//Calculate the number of Device
IF NOT bNumberIsCalculatet THEN
	IF diActualNumberOfDevices < diMaxNumberOfDevices THEN diNumberForThisDevice := diActualNumberOfDevices + 1; bNumberIsCalculatet := TRUE; END_IF 
		diNumberOfTotalDevices := diActualNumberOfDevices + 1;
			FPCalculatet.CLK := TRUE;
				diNumberForThisDevice := LIMIT(0,diNumberForThisDevice,diMaxNumberOfDevices);		
END_IF 
	//Reset when we have a online change
	IF bOnlineChange THEN bOnlineChange := FALSE; END_IF
		IF udiCounterOnlineChange <> udiCounterOnlineChange_CP THEN
			bNumberIsCalculatet := FALSE;
				diNumberForThisDevice := 0;
					diNumberOfTotalDevices := diNumberForThisDevice;
						udiCounterOnlineChange_CP := udiCounterOnlineChange;   
							bOnlineChange := TRUE;	
								FPCalculatet.CLK := FALSE;			
		END_IF  
		
FPCalculatet(CLK:= , Q=> bFPNumberIsCalculatet);

END_FUNCTION_BLOCK

// ---- Persistent Data/FBs Internal/PD Slave/FB_PersistentData_String.TcPOU
{attribute 'hide_all_locals'}
{attribute 'conditionalshow'}
FUNCTION_BLOCK FB_PersistentData_String
VAR_INPUT
	{attribute 'hide'}
	sText								: STRING(255);			//Actual Input Text						
END_VAR
VAR_OUTPUT
	{attribute 'hide'}
	bEventBasedActive					: BOOL;					//Event based saving is active
END_VAR
VAR
	sText_CP							: STRING(255);			//Text to compare the input Text
	fbTaskIndex							: GETCURTASKINDEX;		//Get the Task index
END_VAR

//Creator : Kai Ebensperger
//Company : Lynus AG
//Date : 15.02.2021
//Version : 1.0.0.0

//With this Function we can check if the Value on the Input of the Function ha changed an chan start to saving the persistent Data in Event Based Mode
//Work only with String Fromat
//Max 255 characters

//---------------------------------------------------------------Logic to start the save process---------------------------------------------------------------------------------------

bEventBasedActive := GVL_Persistent_Data.bEventBasedActive;

//After Restart the System set the Variables direct to actual value because they are loadet from the card
fbTaskIndex(index=> );
	IF TwinCAT_SystemInfoVarList._TaskInfo[fbTaskIndex.index].FirstCycle THEN sText_CP := sText; END_IF

IF NOT GVL_Persistent_Data.bBusy AND bEventBasedActive AND MEMCMP(ADR(sText),ADR(sText_CP),SIZEOF(sText_CP)) <> 0 THEN
	GVL_Persistent_Data.bSaveData := TRUE;
		sText_CP := sText;
END_IF

END_FUNCTION_BLOCK

// ---- Sensors/FBs Internal/Temperature/FB_Config_KL320x.TcPOU
{attribute 'conditionalshow'}
FUNCTION_BLOCK FB_Config_KL320x
VAR_INPUT
	{attribute 'hide'}
	eChooseSensorType		: E_ChooseSensortype_KL320x;			//Tel what sensor type is configred on the terminal
	{attribute 'hide'}
	iTimeout				: INT;									//Delay for timeout in seconds
	{attribute 'hide'}
	bWriteConfig			: BOOL;									//Positive edge start the sensor type configuration on the terminal
	{attribute 'hide'}
	bReadConfig				: BOOL;									//Posistive edge read out the actual configuration from the terminal
END_VAR
VAR_OUTPUT
	{attribute 'hide'}
	bConfigModeAktiv		: BOOL;									//True when the configuration mode is active
	{attribute 'hide'}
	bError					: BOOL;									//Error Bit
	{attribute 'hide'}
	b2Wire					: BOOL;									//Terminal is configured in the 2 wire mode
	{attribute 'hide'}
	iRawValueTerminal		: INT;									//Raw value from the terminal when the configuration mode is done
	{attribute 'hide'}
	usiState				: USINT;								//State from the KL320x terminal
	{attribute 'hide'}
	sSensorType				: STRING(50);							//Configured sensortype as string after read out the configuration
END_VAR
VAR
	{attribute 'hide'}
	FP0						: R_TRIG;								//Internal positive edge
	{attribute 'hide'}
	FP1						: R_TRIG;								//Internal positive edge
	{attribute 'hide'}
	timTimout				: TON;									//Timer for timeout
	{attribute 'hide'}
	eStep					: E_Step_Config_Terminal_KL320x;		//Step terminal configuration
	stDataIn		AT%I*	: ST_InputData_KL320x;					//Input Data from the KL320x
	stDataOut		AT%Q*	: ST_OutputData_KL320x;					//Output Data from the KL320x
	{attribute 'hide'}
	bCheck					: BOOL;									//True after the value is writen in the register
END_VAR

//Creator : Kai Ebensperger
//Company : Lynus AG
//Date : 02.06.2021
//Version : 1.0.0.0

//This function block is used to configure a KL3201, KL3202 and KL3204
//Communicate about the input and output Data from the terminal
//Attention : A KL3208 cannot be configured with this function block

(*---------------------------------------------------------------Check the limits of the inputs-------------------------------------------------------------------------------*)

iTimeout := LIMIT(1,iTimeout,10);

(*---------------------------------------------------------------Start the configuration or read out the actual configuration-------------------------------------------------------------------------------*)

FP0(CLK:= bWriteConfig, Q=> );
	FP1(CLK:= bReadConfig, Q=> );

	IF FP0.Q AND NOT bConfigModeAktiv THEN
		eStep := E_Step_Config_Terminal_KL320x.eRegister31DeactivateWriteProtection_KL320x;
	END_IF
		IF FP1.Q AND NOT bConfigModeAktiv THEN
			eStep := E_Step_Config_Terminal_KL320x.eReadConfiguration_KL320x;
		END_IF
	
CASE eStep OF
		
	E_Step_Config_Terminal_KL320x.eInit_KL320x: //Init Step						
										
		iRawValueTerminal := stDataIn.iDataIn;
			usiState := stDataIn.usiState;
				stDataOut.iDataOut := 0;
					stDataOut.usiControl := 0;
						bConfigModeAktiv := FALSE;
							timTimout.IN := FALSE;
								bCheck := FALSE;
			
	E_Step_Config_Terminal_KL320x.eRegister31DeactivateWriteProtection_KL320x: //Deactivate Write protecton on register 31 to write data on other registers			
													
		bConfigModeAktiv := TRUE;
			timTimout.IN := TRUE;
				bError := FALSE;
							
					IF NOT bCheck THEN	
						stDataOut.usiControl.0 := TRUE;
							stDataOut.usiControl.1 := TRUE;
								stDataOut.usiControl.2 := TRUE;
									stDataOut.usiControl.3 := TRUE;
										stDataOut.usiControl.4 := TRUE;
											stDataOut.usiControl.5 := FALSE;				
												stDataOut.usiControl.6 := TRUE;
													stDataOut.usiControl.7 := TRUE;
						END_IF
														
							//Activate the code in register 31
							stDataOut.iDataOut := 16#1235;
		
							//Feedback from the input data from the terminal
							IF stDataIn.iDataIn.0 = FALSE AND
								stDataIn.iDataIn.1 = FALSE AND
									stDataIn.iDataIn.2 = FALSE AND
										stDataIn.iDataIn.3 = FALSE AND
											stDataIn.iDataIn.4 = FALSE AND
												stDataIn.iDataIn.5 = FALSE AND
													stDataIn.iDataIn.6 = FALSE AND
														stDataIn.iDataIn.7 = FALSE AND
															stDataIn.iDataIn.8 = FALSE AND
																stDataIn.iDataIn.9 = FALSE AND
																	stDataIn.iDataIn.10 = FALSE AND
																		stDataIn.iDataIn.11 = FALSE AND
																			stDataIn.iDataIn.12 = FALSE AND
																				stDataIn.iDataIn.13 = FALSE AND
																					stDataIn.iDataIn.14 = FALSE AND
																						stDataIn.iDataIn.15 = FALSE AND
																							stDataIn.usiState = 159 AND
																								stDataOut.iDataOut = 16#1235 THEN
								//Check if the value is writen in register 31
								stDataOut.usiControl.0 := TRUE;
									stDataOut.usiControl.1 := TRUE;
										stDataOut.usiControl.2 := TRUE;
											stDataOut.usiControl.3 := TRUE;
												stDataOut.usiControl.4 := TRUE;
													stDataOut.usiControl.5 := FALSE;				
														stDataOut.usiControl.6 := FALSE;
															stDataOut.usiControl.7 := TRUE;
																bCheck := TRUE;	
																								
							END_IF	
						
							//Feedback from Input data for register access
							IF stDataIn.iDataIn.0 = TRUE AND
								stDataIn.iDataIn.1 = FALSE AND
									stDataIn.iDataIn.2 = TRUE AND
										stDataIn.iDataIn.3 = FALSE AND
											stDataIn.iDataIn.4 = TRUE AND
												stDataIn.iDataIn.5 = TRUE AND
													stDataIn.iDataIn.6 = FALSE AND
														stDataIn.iDataIn.7 = FALSE AND
															stDataIn.iDataIn.8 = FALSE AND
																stDataIn.iDataIn.9 = TRUE AND
																	stDataIn.iDataIn.10 = FALSE AND
																		stDataIn.iDataIn.11 = FALSE AND
																			stDataIn.iDataIn.12 = TRUE AND
																				stDataIn.iDataIn.13 = FALSE AND
																					stDataIn.iDataIn.14 = FALSE AND
																						stDataIn.iDataIn.15 = FALSE AND
																							stDataIn.usiState = 159 THEN 
								eStep := E_Step_Config_Terminal_KL320x.eChooseSensorType_KL320x;
							END_IF
					
	E_Step_Config_Terminal_KL320x.eChooseSensorType_KL320x: //Choose sensor the type	
						
		bCheck := FALSE;
	
			//PT100
			IF eChooseSensorType = E_ChooseSensortype_KL320x.ePT100_KL320x THEN
				eStep :=  E_Step_Config_Terminal_KL320x.ePT100Config_KL320x;
			END_IF								
									
			//PT1000
			IF eChooseSensorType = E_ChooseSensortype_KL320x.ePT1000_KL320x THEN
				eStep :=  E_Step_Config_Terminal_KL320x.ePT1000Config_KL320x;
			END_IF
		
			//PT1000 2 wire !!Not possible for KL3204!!
			IF eChooseSensorType = E_ChooseSensortype_KL320x.ePT10002Leiter_KL320x THEN
				eStep :=  E_Step_Config_Terminal_KL320x.ePT10002WireConfig_KL320x;
			END_IF
							
			//PT500
			IF eChooseSensorType = E_ChooseSensortype_KL320x.ePT500_KL320x THEN
				eStep :=  E_Step_Config_Terminal_KL320x.ePT500Config_KL320x;
			END_IF
								
			//PT200
			IF eChooseSensorType = E_ChooseSensortype_KL320x.ePT200_KL320x THEN
				eStep :=  E_Step_Config_Terminal_KL320x.ePT200Config_KL320x;
			END_IF
								
			//NI100
			IF eChooseSensorType = E_ChooseSensortype_KL320x.eNI100_KL320x THEN
				eStep :=  E_Step_Config_Terminal_KL320x.eNI100Config_KL320x;
			END_IF
								
			//NI1000
			IF eChooseSensorType = E_ChooseSensortype_KL320x.eNI1000_KL320x THEN
				eStep :=  E_Step_Config_Terminal_KL320x.eNI1000Config_KL320x;
			END_IF
		
			//NI120
			IF eChooseSensorType = E_ChooseSensortype_KL320x.eNI120_KL320x THEN
				eStep :=  E_Step_Config_Terminal_KL320x.eNI120Config_KL320x;
			END_IF
		
			//Resistor from 10 Ohm to 5 kOhm
			IF eChooseSensorType = E_ChooseSensortype_KL320x.eResistor10Ohm5000Ohm_KL320x THEN
				eStep :=  E_Step_Config_Terminal_KL320x.e10Ohm5000OhmConfig_KL320x;
			END_IF
								
			//Resistor from  10 Ohm to 1,2kOhm
			IF eChooseSensorType = E_ChooseSensortype_KL320x.eResistor10Ohm1200Ohm_KL320x THEN
				eStep := E_Step_Config_Terminal_KL320x.e10Ohm1200OhmConfig_KL320x;
			END_IF
	
	E_Step_Config_Terminal_KL320x.ePT100Config_KL320x: //Register 32 for PT100 configuration	
							
		IF NOT bCheck THEN					
			stDataOut.usiControl.0 := FALSE;
				stDataOut.usiControl.1 := FALSE;
					stDataOut.usiControl.2 := FALSE;
						stDataOut.usiControl.3 := FALSE;
							stDataOut.usiControl.4 := FALSE;
								stDataOut.usiControl.5 := TRUE;				
									stDataOut.usiControl.6 := TRUE;
										stDataOut.usiControl.7 := TRUE;
		END_IF
							
			//Code for PT100
			stDataOut.iDataOut := 16#0106;
								
				//Feedback from the input data from the terminal
				IF stDataIn.iDataIn.0 = FALSE AND
					stDataIn.iDataIn.1 = FALSE AND
						stDataIn.iDataIn.2 = FALSE AND
							stDataIn.iDataIn.3 = FALSE AND
								stDataIn.iDataIn.4 = FALSE AND
									stDataIn.iDataIn.5 = FALSE AND
										stDataIn.iDataIn.6 = FALSE AND
											stDataIn.iDataIn.7 = FALSE AND
												stDataIn.iDataIn.8 = FALSE AND
													stDataIn.iDataIn.9 = FALSE AND
														stDataIn.iDataIn.10 = FALSE AND
															stDataIn.iDataIn.11 = FALSE AND
																stDataIn.iDataIn.12 = FALSE AND
																	stDataIn.iDataIn.13 = FALSE AND
																		stDataIn.iDataIn.14 = FALSE AND
																			stDataIn.iDataIn.15 = FALSE AND
																				stDataIn.usiState = 160 AND
																					stDataOut.iDataOut = 16#0106 THEN
				//Check if the value is writen in register 32
				stDataOut.usiControl.0 := FALSE;
					stDataOut.usiControl.1 := FALSE;
						stDataOut.usiControl.2 := FALSE;
							stDataOut.usiControl.3 := FALSE;
								stDataOut.usiControl.4 := FALSE;
									stDataOut.usiControl.5 := TRUE;				
										stDataOut.usiControl.6 := FALSE;
											stDataOut.usiControl.7 := TRUE;
												bCheck := TRUE;	
																									
				END_IF	
				
					//Feedback from Input data for register access			
					IF stDataIn.iDataIn.0 = FALSE AND
						stDataIn.iDataIn.1 = TRUE AND
							stDataIn.iDataIn.2 = TRUE AND
								stDataIn.iDataIn.3 = FALSE AND
									stDataIn.iDataIn.4 = FALSE AND
										stDataIn.iDataIn.5 = FALSE AND
											stDataIn.iDataIn.6 = FALSE AND
												stDataIn.iDataIn.7 = FALSE AND
													stDataIn.iDataIn.8 = TRUE AND
														stDataIn.iDataIn.9 = FALSE AND
															stDataIn.iDataIn.10 = FALSE AND
																stDataIn.iDataIn.11 = FALSE AND
																	stDataIn.iDataIn.12 = FALSE AND
																		stDataIn.iDataIn.13 = FALSE AND
																			stDataIn.iDataIn.14 = FALSE AND
																				stDataIn.iDataIn.15 = FALSE AND
																					stDataIn.usiState = 160 THEN 
						eStep := E_Step_Config_Terminal_KL320x.eControlByteNull_KL320x;
					END_IF																	
						
	E_Step_Config_Terminal_KL320x.ePT1000Config_KL320x: //Register 32 for PT1000 configuration			
									
		IF NOT bCheck THEN
			stDataOut.usiControl.0 := FALSE;
				stDataOut.usiControl.1 := FALSE;
					stDataOut.usiControl.2 := FALSE;
						stDataOut.usiControl.3 := FALSE;
							stDataOut.usiControl.4 := FALSE;
								stDataOut.usiControl.5 := TRUE;				
									stDataOut.usiControl.6 := TRUE;
										stDataOut.usiControl.7 := TRUE;
		END_IF
							
			//Code for PT1000
			stDataOut.iDataOut := 16#2106;
									
				//Feedback from the input data from the terminal
				IF stDataIn.iDataIn.0 = FALSE AND
					stDataIn.iDataIn.1 = FALSE AND
						stDataIn.iDataIn.2 = FALSE AND
							stDataIn.iDataIn.3 = FALSE AND
								stDataIn.iDataIn.4 = FALSE AND
									stDataIn.iDataIn.5 = FALSE AND
										stDataIn.iDataIn.6 = FALSE AND
											stDataIn.iDataIn.7 = FALSE AND
												stDataIn.iDataIn.8 = FALSE AND
													stDataIn.iDataIn.9 = FALSE AND
														stDataIn.iDataIn.10 = FALSE AND
															stDataIn.iDataIn.11 = FALSE AND
																stDataIn.iDataIn.12 = FALSE AND
																	stDataIn.iDataIn.13 = FALSE AND
																		stDataIn.iDataIn.14 = FALSE AND
																			stDataIn.iDataIn.15 = FALSE AND
																				stDataIn.usiState = 160 AND
																					stDataOut.iDataOut = 16#2106 THEN
				//Check if the value is writen in register 32
				stDataOut.usiControl.0 := FALSE;
					stDataOut.usiControl.1 := FALSE;
						stDataOut.usiControl.2 := FALSE;
							stDataOut.usiControl.3 := FALSE;
								stDataOut.usiControl.4 := FALSE;
									stDataOut.usiControl.5 := TRUE;				
										stDataOut.usiControl.6 := FALSE;
											stDataOut.usiControl.7 := TRUE;
												bCheck := TRUE;	
																										
				END_IF	
					
					//Feedback from Input data for register access				
					IF stDataIn.iDataIn.0 = FALSE AND
						stDataIn.iDataIn.1 = TRUE AND
							stDataIn.iDataIn.2 = TRUE AND
								stDataIn.iDataIn.3 = FALSE AND
									stDataIn.iDataIn.4 = FALSE AND
										stDataIn.iDataIn.5 = FALSE AND
											stDataIn.iDataIn.6 = FALSE AND
												stDataIn.iDataIn.7 = FALSE AND
													stDataIn.iDataIn.8 = TRUE AND
														stDataIn.iDataIn.9 = FALSE AND
															stDataIn.iDataIn.10 = FALSE AND
																stDataIn.iDataIn.11 = FALSE AND
																	stDataIn.iDataIn.12 = FALSE AND
																		stDataIn.iDataIn.13 = TRUE AND
																			stDataIn.iDataIn.14 = FALSE AND
																				stDataIn.iDataIn.15 = FALSE AND
																					stDataIn.usiState = 160 THEN 
						eStep := E_Step_Config_Terminal_KL320x.eControlByteNull_KL320x;
					END_IF							
												
	E_Step_Config_Terminal_KL320x.ePT10002WireConfig_KL320x: //Register 32 for PT1000 configuration with 2 wire technic !!!Not work with the KL3204 terminal!!!
	
		IF NOT bCheck THEN
			stDataOut.usiControl.0 := FALSE;
				stDataOut.usiControl.1 := FALSE;
					stDataOut.usiControl.2 := FALSE;
						stDataOut.usiControl.3 := FALSE;
							stDataOut.usiControl.4 := FALSE;
								stDataOut.usiControl.5 := TRUE;				
									stDataOut.usiControl.6 := TRUE;
										stDataOut.usiControl.7 := TRUE;
		END_IF
										
			//Code for PT1000 2 wire technic
			stDataOut.iDataOut := 16#2506;
										
				//Feedback from the input data from the terminal
				IF stDataIn.iDataIn.0 = FALSE AND
					stDataIn.iDataIn.1 = FALSE AND
						stDataIn.iDataIn.2 = FALSE AND
							stDataIn.iDataIn.3 = FALSE AND
								stDataIn.iDataIn.4 = FALSE AND
									stDataIn.iDataIn.5 = FALSE AND
										stDataIn.iDataIn.6 = FALSE AND
											stDataIn.iDataIn.7 = FALSE AND
												stDataIn.iDataIn.8 = FALSE AND
													stDataIn.iDataIn.9 = FALSE AND
														stDataIn.iDataIn.10 = FALSE AND
															stDataIn.iDataIn.11 = FALSE AND
																stDataIn.iDataIn.12 = FALSE AND
																	stDataIn.iDataIn.13 = FALSE AND
																		stDataIn.iDataIn.14 = FALSE AND
																			stDataIn.iDataIn.15 = FALSE AND
																				stDataIn.usiState = 160 AND
																					stDataOut.iDataOut = 16#2506 THEN
				//Check if the value is writen in register 32
				stDataOut.usiControl.0 := FALSE;
					stDataOut.usiControl.1 := FALSE;
						stDataOut.usiControl.2 := FALSE;
							stDataOut.usiControl.3 := FALSE;
								stDataOut.usiControl.4 := FALSE;
									stDataOut.usiControl.5 := TRUE;				
										stDataOut.usiControl.6 := FALSE;
											stDataOut.usiControl.7 := TRUE;
												bCheck := TRUE;	
																											
				END_IF	
						
					//Feedback from Input data for register access					
					IF stDataIn.iDataIn.0 = FALSE AND
						stDataIn.iDataIn.1 = TRUE AND
							stDataIn.iDataIn.2 = TRUE AND
								stDataIn.iDataIn.3 = FALSE AND
									stDataIn.iDataIn.4 = FALSE AND
										stDataIn.iDataIn.5 = FALSE AND
											stDataIn.iDataIn.6 = FALSE AND
												stDataIn.iDataIn.7 = FALSE AND
													stDataIn.iDataIn.8 = TRUE AND
														stDataIn.iDataIn.9 = FALSE AND
															stDataIn.iDataIn.10 = TRUE AND
																stDataIn.iDataIn.11 = FALSE AND
																	stDataIn.iDataIn.12 = FALSE AND
																		stDataIn.iDataIn.13 = TRUE AND
																			stDataIn.iDataIn.14 = FALSE AND
																				stDataIn.iDataIn.15 = FALSE AND
																					stDataIn.usiState = 160 THEN 
						eStep := E_Step_Config_Terminal_KL320x.eControlByteNull_KL320x;
					END_IF	
	
	E_Step_Config_Terminal_KL320x.ePT500Config_KL320x:	//Register 32 for PT500 configuration
								
		IF NOT bCheck THEN
			stDataOut.usiControl.0 := FALSE;
				stDataOut.usiControl.1 := FALSE;
					stDataOut.usiControl.2 := FALSE;
						stDataOut.usiControl.3 := FALSE;
							stDataOut.usiControl.4 := FALSE;
								stDataOut.usiControl.5 := TRUE;				
									stDataOut.usiControl.6 := TRUE;
										stDataOut.usiControl.7 := TRUE;
		END_IF
									
			//Code for PT500
			stDataOut.iDataOut := 16#3106;
										
				//Feedback from the input data from the terminal
				IF stDataIn.iDataIn.0 = FALSE AND
					stDataIn.iDataIn.1 = FALSE AND
						stDataIn.iDataIn.2 = FALSE AND
							stDataIn.iDataIn.3 = FALSE AND
								stDataIn.iDataIn.4 = FALSE AND
									stDataIn.iDataIn.5 = FALSE AND
										stDataIn.iDataIn.6 = FALSE AND
											stDataIn.iDataIn.7 = FALSE AND
												stDataIn.iDataIn.8 = FALSE AND
													stDataIn.iDataIn.9 = FALSE AND
														stDataIn.iDataIn.10 = FALSE AND
															stDataIn.iDataIn.11 = FALSE AND
																stDataIn.iDataIn.12 = FALSE AND
																	stDataIn.iDataIn.13 = FALSE AND
																		stDataIn.iDataIn.14 = FALSE AND
																			stDataIn.iDataIn.15 = FALSE AND
																				stDataIn.usiState = 160 AND
																					stDataOut.iDataOut = 16#3106 THEN
				//Check if the value is writen in register 32
				stDataOut.usiControl.0 := FALSE;
					stDataOut.usiControl.1 := FALSE;
						stDataOut.usiControl.2 := FALSE;
							stDataOut.usiControl.3 := FALSE;
								stDataOut.usiControl.4 := FALSE;
									stDataOut.usiControl.5 := TRUE;				
										stDataOut.usiControl.6 := FALSE;
											stDataOut.usiControl.7 := TRUE;
												bCheck := TRUE;	
				END_IF	
					
					//Feedback from Input data for register access						
					IF stDataIn.iDataIn.0 = FALSE AND
						stDataIn.iDataIn.1 = TRUE AND
							stDataIn.iDataIn.2 = TRUE AND
								stDataIn.iDataIn.3 = FALSE AND
									stDataIn.iDataIn.4 = FALSE AND
										stDataIn.iDataIn.5 = FALSE AND
											stDataIn.iDataIn.6 = FALSE AND
												stDataIn.iDataIn.7 = FALSE AND
													stDataIn.iDataIn.8 = TRUE AND
														stDataIn.iDataIn.9 = FALSE AND
															stDataIn.iDataIn.10 = FALSE AND
																stDataIn.iDataIn.11 = FALSE AND
																	stDataIn.iDataIn.12 = TRUE AND
																		stDataIn.iDataIn.13 = TRUE AND
																			stDataIn.iDataIn.14 = FALSE AND
																				stDataIn.iDataIn.15 = FALSE AND
																					stDataIn.usiState = 160 THEN 
						eStep := E_Step_Config_Terminal_KL320x.eControlByteNull_KL320x;
					END_IF
	
	E_Step_Config_Terminal_KL320x.ePT200Config_KL320x :	//Register 32 for PT200 configuration
	
		IF NOT bCheck THEN
			stDataOut.usiControl.0 := FALSE;
				stDataOut.usiControl.1 := FALSE;
					stDataOut.usiControl.2 := FALSE;
						stDataOut.usiControl.3 := FALSE;
							stDataOut.usiControl.4 := FALSE;
								stDataOut.usiControl.5 := TRUE;				
									stDataOut.usiControl.6 := TRUE;
										stDataOut.usiControl.7 := TRUE;
		END_IF
									
			//Code for PT200
			stDataOut.iDataOut := 16#4106;
											
				//Feedback from the input data from the terminal
				IF stDataIn.iDataIn.0 = FALSE AND
					stDataIn.iDataIn.1 = FALSE AND
						stDataIn.iDataIn.2 = FALSE AND
							stDataIn.iDataIn.3 = FALSE AND
								stDataIn.iDataIn.4 = FALSE AND
									stDataIn.iDataIn.5 = FALSE AND
										stDataIn.iDataIn.6 = FALSE AND
											stDataIn.iDataIn.7 = FALSE AND
												stDataIn.iDataIn.8 = FALSE AND
													stDataIn.iDataIn.9 = FALSE AND
														stDataIn.iDataIn.10 = FALSE AND
															stDataIn.iDataIn.11 = FALSE AND
																stDataIn.iDataIn.12 = FALSE AND
																	stDataIn.iDataIn.13 = FALSE AND
																		stDataIn.iDataIn.14 = FALSE AND
																			stDataIn.iDataIn.15 = FALSE AND
																				stDataIn.usiState = 160 AND
																					stDataOut.iDataOut = 16#4106 THEN
				//Check if the value is writen in register 32
				stDataOut.usiControl.0 := FALSE;
					stDataOut.usiControl.1 := FALSE;
						stDataOut.usiControl.2 := FALSE;
							stDataOut.usiControl.3 := FALSE;
								stDataOut.usiControl.4 := FALSE;
									stDataOut.usiControl.5 := TRUE;				
										stDataOut.usiControl.6 := FALSE;
											stDataOut.usiControl.7 := TRUE;
												bCheck := TRUE;	
				END_IF	
						
					//Feedback from Input data for register access						
					IF stDataIn.iDataIn.0 = FALSE AND
							stDataIn.iDataIn.1 = TRUE AND
								stDataIn.iDataIn.2 = TRUE AND
									stDataIn.iDataIn.3 = FALSE AND
										stDataIn.iDataIn.4 = FALSE AND
											stDataIn.iDataIn.5 = FALSE AND
												stDataIn.iDataIn.6 = FALSE AND
													stDataIn.iDataIn.7 = FALSE AND
														stDataIn.iDataIn.8 = TRUE AND
															stDataIn.iDataIn.9 = FALSE AND
																stDataIn.iDataIn.10 = FALSE AND
																	stDataIn.iDataIn.11 = FALSE AND
																		stDataIn.iDataIn.12 = FALSE AND
																			stDataIn.iDataIn.13 = FALSE AND
																				stDataIn.iDataIn.14 = TRUE AND
																					stDataIn.iDataIn.15 = FALSE AND
																						stDataIn.usiState = 160 THEN 
						eStep := E_Step_Config_Terminal_KL320x.eControlByteNull_KL320x;
					END_IF
	
	E_Step_Config_Terminal_KL320x.eNI100Config_KL320x:	//Register 32 for NI100 Kcnfigurieren
	
		IF NOT bCheck THEN
			stDataOut.usiControl.0 := FALSE;
				stDataOut.usiControl.1 := FALSE;
					stDataOut.usiControl.2 := FALSE;
						stDataOut.usiControl.3 := FALSE;
							stDataOut.usiControl.4 := FALSE;
								stDataOut.usiControl.5 := TRUE;				
									stDataOut.usiControl.6 := TRUE;
										stDataOut.usiControl.7 := TRUE;
		END_IF
									
			//Code for NI100
			stDataOut.iDataOut := 16#1106;
										
				//Feedback from the input data from the terminal
				IF stDataIn.iDataIn.0 = FALSE AND
					stDataIn.iDataIn.1 = FALSE AND
						stDataIn.iDataIn.2 = FALSE AND
							stDataIn.iDataIn.3 = FALSE AND
								stDataIn.iDataIn.4 = FALSE AND
									stDataIn.iDataIn.5 = FALSE AND
										stDataIn.iDataIn.6 = FALSE AND
											stDataIn.iDataIn.7 = FALSE AND
												stDataIn.iDataIn.8 = FALSE AND
													stDataIn.iDataIn.9 = FALSE AND
														stDataIn.iDataIn.10 = FALSE AND
															stDataIn.iDataIn.11 = FALSE AND
																stDataIn.iDataIn.12 = FALSE AND
																	stDataIn.iDataIn.13 = FALSE AND
																		stDataIn.iDataIn.14 = FALSE AND
																			stDataIn.iDataIn.15 = FALSE AND
																				stDataIn.usiState = 160 AND
																					stDataOut.iDataOut = 16#1106 THEN
				//Check if the value is writen in register 32
				stDataOut.usiControl.0 := FALSE;
					stDataOut.usiControl.1 := FALSE;
						stDataOut.usiControl.2 := FALSE;
							stDataOut.usiControl.3 := FALSE;
								stDataOut.usiControl.4 := FALSE;
									stDataOut.usiControl.5 := TRUE;				
										stDataOut.usiControl.6 := FALSE;
											stDataOut.usiControl.7 := TRUE;
												bCheck := TRUE;	
				END_IF	
						
					//Feedback from Input data for register access					
					IF stDataIn.iDataIn.0 = FALSE AND
						stDataIn.iDataIn.1 = TRUE AND
							stDataIn.iDataIn.2 = TRUE AND
								stDataIn.iDataIn.3 = FALSE AND
									stDataIn.iDataIn.4 = FALSE AND
										stDataIn.iDataIn.5 = FALSE AND
											stDataIn.iDataIn.6 = FALSE AND
												stDataIn.iDataIn.7 = FALSE AND
													stDataIn.iDataIn.8 = TRUE AND
														stDataIn.iDataIn.9 = FALSE AND
															stDataIn.iDataIn.10 = FALSE AND
																stDataIn.iDataIn.11 = FALSE AND
																	stDataIn.iDataIn.12 = TRUE AND
																		stDataIn.iDataIn.13 = FALSE AND
																			stDataIn.iDataIn.14 = FALSE AND
																				stDataIn.iDataIn.15 = FALSE AND
																					stDataIn.usiState = 160 THEN 
						eStep := E_Step_Config_Terminal_KL320x.eControlByteNull_KL320x;
					END_IF
	
	E_Step_Config_Terminal_KL320x.eNI1000Config_KL320x:	//Register 32 for NI1000 configurieren
	
		IF NOT bCheck THEN
			stDataOut.usiControl.0 := FALSE;
				stDataOut.usiControl.1 := FALSE;
					stDataOut.usiControl.2 := FALSE;
						stDataOut.usiControl.3 := FALSE;
							stDataOut.usiControl.4 := FALSE;
								stDataOut.usiControl.5 := TRUE;				
									stDataOut.usiControl.6 := TRUE;
										stDataOut.usiControl.7 := TRUE;
		END_IF
									
			//Code for NI1000
			stDataOut.iDataOut := 16#5106;
											
				//Feedback from the input data from the terminal
				IF stDataIn.iDataIn.0 = FALSE AND
					stDataIn.iDataIn.1 = FALSE AND
						stDataIn.iDataIn.2 = FALSE AND
							stDataIn.iDataIn.3 = FALSE AND
								stDataIn.iDataIn.4 = FALSE AND
									stDataIn.iDataIn.5 = FALSE AND
										stDataIn.iDataIn.6 = FALSE AND
											stDataIn.iDataIn.7 = FALSE AND
												stDataIn.iDataIn.8 = FALSE AND
													stDataIn.iDataIn.9 = FALSE AND
														stDataIn.iDataIn.10 = FALSE AND
															stDataIn.iDataIn.11 = FALSE AND
																stDataIn.iDataIn.12 = FALSE AND
																	stDataIn.iDataIn.13 = FALSE AND
																		stDataIn.iDataIn.14 = FALSE AND
																			stDataIn.iDataIn.15 = FALSE AND
																				stDataIn.usiState = 160 AND
																					stDataOut.iDataOut = 16#5106 THEN
				//Check if the value is writen in register 32
				stDataOut.usiControl.0 := FALSE;
					stDataOut.usiControl.1 := FALSE;
						stDataOut.usiControl.2 := FALSE;
							stDataOut.usiControl.3 := FALSE;
								stDataOut.usiControl.4 := FALSE;
									stDataOut.usiControl.5 := TRUE;				
										stDataOut.usiControl.6 := FALSE;
											stDataOut.usiControl.7 := TRUE;
												bCheck := TRUE;	
				END_IF	
						
					//Feedback from Input data for register access							
					IF stDataIn.iDataIn.0 = FALSE AND
						stDataIn.iDataIn.1 = TRUE AND
							stDataIn.iDataIn.2 = TRUE AND
								stDataIn.iDataIn.3 = FALSE AND
									stDataIn.iDataIn.4 = FALSE AND
										stDataIn.iDataIn.5 = FALSE AND
											stDataIn.iDataIn.6 = FALSE AND
												stDataIn.iDataIn.7 = FALSE AND
													stDataIn.iDataIn.8 = TRUE AND
														stDataIn.iDataIn.9 = FALSE AND
															stDataIn.iDataIn.10 = FALSE AND
																stDataIn.iDataIn.11 = FALSE AND
																	stDataIn.iDataIn.12 = TRUE AND
																		stDataIn.iDataIn.13 = FALSE AND
																			stDataIn.iDataIn.14 = TRUE AND
																				stDataIn.iDataIn.15 = FALSE AND
																					stDataIn.usiState = 160 THEN 
						eStep := E_Step_Config_Terminal_KL320x.eControlByteNull_KL320x;
					END_IF
	
	E_Step_Config_Terminal_KL320x.eNI120Config_KL320x:	//Register 32 for NI120 configurieren
	
		IF NOT bCheck THEN
			stDataOut.usiControl.0 := FALSE;
				stDataOut.usiControl.1 := FALSE;
					stDataOut.usiControl.2 := FALSE;
						stDataOut.usiControl.3 := FALSE;
							stDataOut.usiControl.4 := FALSE;
								stDataOut.usiControl.5 := TRUE;				
									stDataOut.usiControl.6 := TRUE;
										stDataOut.usiControl.7 := TRUE;
		END_IF
									
			//Code for NI120
			stDataOut.iDataOut := 16#6106;
										
				//Feedback from the input data from the terminal
				IF stDataIn.iDataIn.0 = FALSE AND
					stDataIn.iDataIn.1 = FALSE AND
						stDataIn.iDataIn.2 = FALSE AND
							stDataIn.iDataIn.3 = FALSE AND
								stDataIn.iDataIn.4 = FALSE AND
									stDataIn.iDataIn.5 = FALSE AND
										stDataIn.iDataIn.6 = FALSE AND
											stDataIn.iDataIn.7 = FALSE AND
												stDataIn.iDataIn.8 = FALSE AND
													stDataIn.iDataIn.9 = FALSE AND
														stDataIn.iDataIn.10 = FALSE AND
															stDataIn.iDataIn.11 = FALSE AND
																stDataIn.iDataIn.12 = FALSE AND
																	stDataIn.iDataIn.13 = FALSE AND
																		stDataIn.iDataIn.14 = FALSE AND
																			stDataIn.iDataIn.15 = FALSE AND
																				stDataIn.usiState = 160 AND
																					stDataOut.iDataOut = 16#6106 THEN
				//Check if the value is writen in register 32
				stDataOut.usiControl.0 := FALSE;
					stDataOut.usiControl.1 := FALSE;
						stDataOut.usiControl.2 := FALSE;
							stDataOut.usiControl.3 := FALSE;
								stDataOut.usiControl.4 := FALSE;
									stDataOut.usiControl.5 := TRUE;				
										stDataOut.usiControl.6 := FALSE;
											stDataOut.usiControl.7 := TRUE;
												bCheck := TRUE;	
				END_IF	
					
					//Feedback from Input data for register access					
					IF stDataIn.iDataIn.0 = FALSE AND
						stDataIn.iDataIn.1 = TRUE AND
							stDataIn.iDataIn.2 = TRUE AND
								stDataIn.iDataIn.3 = FALSE AND
									stDataIn.iDataIn.4 = FALSE AND
										stDataIn.iDataIn.5 = FALSE AND
											stDataIn.iDataIn.6 = FALSE AND
												stDataIn.iDataIn.7 = FALSE AND
													stDataIn.iDataIn.8 = TRUE AND
														stDataIn.iDataIn.9 = FALSE AND
															stDataIn.iDataIn.10 = FALSE AND
																stDataIn.iDataIn.11 = FALSE AND
																	stDataIn.iDataIn.12 = FALSE AND
																		stDataIn.iDataIn.13 = TRUE AND
																			stDataIn.iDataIn.14 = TRUE AND
																				stDataIn.iDataIn.15 = FALSE AND
																					stDataIn.usiState = 160 THEN 
						eStep := E_Step_Config_Terminal_KL320x.eControlByteNull_KL320x;
					END_IF
	
	E_Step_Config_Terminal_KL320x.e10Ohm5000OhmConfig_KL320x:	//Register 32 for resistor from 10Ohm to 5000Ohm configuration
	
		IF NOT bCheck THEN
			stDataOut.usiControl.0 := FALSE;
				stDataOut.usiControl.1 := FALSE;
					stDataOut.usiControl.2 := FALSE;
						stDataOut.usiControl.3 := FALSE;
							stDataOut.usiControl.4 := FALSE;
								stDataOut.usiControl.5 := TRUE;				
									stDataOut.usiControl.6 := TRUE;
										stDataOut.usiControl.7 := TRUE;
		END_IF
									
			//Code for resistor from 10Ohm to 5000Ohm
			stDataOut.iDataOut := UINT_TO_INT(16#E106);
											
				//Feedback from the input data from the terminal
				IF stDataIn.iDataIn.0 = FALSE AND
					stDataIn.iDataIn.1 = FALSE AND
						stDataIn.iDataIn.2 = FALSE AND
							stDataIn.iDataIn.3 = FALSE AND
								stDataIn.iDataIn.4 = FALSE AND
									stDataIn.iDataIn.5 = FALSE AND
										stDataIn.iDataIn.6 = FALSE AND
											stDataIn.iDataIn.7 = FALSE AND
												stDataIn.iDataIn.8 = FALSE AND
													stDataIn.iDataIn.9 = FALSE AND
														stDataIn.iDataIn.10 = FALSE AND
															stDataIn.iDataIn.11 = FALSE AND
																stDataIn.iDataIn.12 = FALSE AND
																	stDataIn.iDataIn.13 = FALSE AND
																		stDataIn.iDataIn.14 = FALSE AND
																			stDataIn.iDataIn.15 = FALSE AND
																				stDataIn.usiState = 160 AND
																					stDataOut.iDataOut = UINT_TO_INT(16#E106) THEN
											
				//Check if the value is writen in register 32
				stDataOut.usiControl.0 := FALSE;
					stDataOut.usiControl.1 := FALSE;
						stDataOut.usiControl.2 := FALSE;
							stDataOut.usiControl.3 := FALSE;
								stDataOut.usiControl.4 := FALSE;
									stDataOut.usiControl.5 := TRUE;				
										stDataOut.usiControl.6 := FALSE;
											stDataOut.usiControl.7 := TRUE;
												bCheck := TRUE;	
				END_IF	
							
					//Feedback from Input data for register access					
					IF stDataIn.iDataIn.0 = FALSE AND
						stDataIn.iDataIn.1 = TRUE AND
							stDataIn.iDataIn.2 = TRUE AND
								stDataIn.iDataIn.3 = FALSE AND
									stDataIn.iDataIn.4 = FALSE AND
										stDataIn.iDataIn.5 = FALSE AND
											stDataIn.iDataIn.6 = FALSE AND
												stDataIn.iDataIn.7 = FALSE AND
													stDataIn.iDataIn.8 = TRUE AND
														stDataIn.iDataIn.9 = FALSE AND
															stDataIn.iDataIn.10 = FALSE AND
																stDataIn.iDataIn.11 = FALSE AND
																	stDataIn.iDataIn.12 = FALSE AND
																		stDataIn.iDataIn.13 = TRUE AND
																			stDataIn.iDataIn.14 = TRUE AND
																				stDataIn.iDataIn.15 = TRUE AND
																					stDataIn.usiState = 160 THEN 
						eStep := E_Step_Config_Terminal_KL320x.eControlByteNull_KL320x;
					END_IF
	
	E_Step_Config_Terminal_KL320x.e10Ohm1200OhmConfig_KL320x:	//Register 32 for resistor from 10Ohm to 1200Ohm configuration
	
		IF NOT bCheck THEN
			stDataOut.usiControl.0 := FALSE;
				stDataOut.usiControl.1 := FALSE;
					stDataOut.usiControl.2 := FALSE;
						stDataOut.usiControl.3 := FALSE;
							stDataOut.usiControl.4 := FALSE;
								stDataOut.usiControl.5 := TRUE;				
									stDataOut.usiControl.6 := TRUE;
										stDataOut.usiControl.7 := TRUE;
		END_IF
									
			//Code for resistor from 10Ohm to 1200Ohm
			stDataOut.iDataOut := UINT_TO_INT(16#F106);
											
				//Feedback from the input data from the terminal
				IF stDataIn.iDataIn.0 = FALSE AND
					stDataIn.iDataIn.1 = FALSE AND
						stDataIn.iDataIn.2 = FALSE AND
							stDataIn.iDataIn.3 = FALSE AND
								stDataIn.iDataIn.4 = FALSE AND
									stDataIn.iDataIn.5 = FALSE AND
										stDataIn.iDataIn.6 = FALSE AND
											stDataIn.iDataIn.7 = FALSE AND
												stDataIn.iDataIn.8 = FALSE AND
													stDataIn.iDataIn.9 = FALSE AND
														stDataIn.iDataIn.10 = FALSE AND
															stDataIn.iDataIn.11 = FALSE AND
																stDataIn.iDataIn.12 = FALSE AND
																	stDataIn.iDataIn.13 = FALSE AND
																		stDataIn.iDataIn.14 = FALSE AND
																			stDataIn.iDataIn.15 = FALSE AND
																				stDataIn.usiState = 160 AND
																					stDataOut.iDataOut = UINT_TO_INT(16#F106) THEN
											
				//Check if the value is writen in register 32
				stDataOut.usiControl.0 := FALSE;
					stDataOut.usiControl.1 := FALSE;
						stDataOut.usiControl.2 := FALSE;
							stDataOut.usiControl.3 := FALSE;
								stDataOut.usiControl.4 := FALSE;
									stDataOut.usiControl.5 := TRUE;				
										stDataOut.usiControl.6 := FALSE;
											stDataOut.usiControl.7 := TRUE;
												bCheck := TRUE;	
				END_IF	
							
					//Feedback from Input data for register access					
					IF stDataIn.iDataIn.0 = FALSE AND
						stDataIn.iDataIn.1 = TRUE AND
							stDataIn.iDataIn.2 = TRUE AND
								stDataIn.iDataIn.3 = FALSE AND
									stDataIn.iDataIn.4 = FALSE AND
										stDataIn.iDataIn.5 = FALSE AND
											stDataIn.iDataIn.6 = FALSE AND
												stDataIn.iDataIn.7 = FALSE AND
													stDataIn.iDataIn.8 = TRUE AND
														stDataIn.iDataIn.9 = FALSE AND
															stDataIn.iDataIn.10 = FALSE AND
																stDataIn.iDataIn.11 = FALSE AND
																	stDataIn.iDataIn.12 = TRUE AND
																		stDataIn.iDataIn.13 = TRUE AND
																			stDataIn.iDataIn.14 = TRUE AND
																				stDataIn.iDataIn.15 = TRUE AND
																					stDataIn.usiState = 160 THEN 
						eStep := E_Step_Config_Terminal_KL320x.eControlByteNull_KL320x;
					END_IF
						
	E_Step_Config_Terminal_KL320x.eControlByteNull_KL320x:	//Set the control Byte to 0
	
		bCheck := FALSE;	
			stDataOut.usiControl := 0;
				eStep := E_Step_Config_Terminal_KL320x.eRegister31ActivateWriteProtection_KL320x;
	
	E_Step_Config_Terminal_KL320x.eRegister31ActivateWriteProtection_KL320x:	//Register 31 activate write protection
	
		IF NOT bCheck THEN
			stDataOut.usiControl.0 := TRUE;
				stDataOut.usiControl.1 := TRUE;
					stDataOut.usiControl.2 := TRUE;
						stDataOut.usiControl.3 := TRUE;
							stDataOut.usiControl.4 := TRUE;
								stDataOut.usiControl.5 := FALSE;				
									stDataOut.usiControl.6 := TRUE;
										stDataOut.usiControl.7 := TRUE;
		END_IF
			
			//Activate the code in Register 31
			stDataOut.iDataOut := 16#0000;
							
				//Feedback from the input data from the terminal
				IF stDataIn.iDataIn.0 = FALSE AND
					stDataIn.iDataIn.1 = FALSE AND
						stDataIn.iDataIn.2 = FALSE AND
							stDataIn.iDataIn.3 = FALSE AND
								stDataIn.iDataIn.4 = FALSE AND
									stDataIn.iDataIn.5 = FALSE AND
										stDataIn.iDataIn.6 = FALSE AND
											stDataIn.iDataIn.7 = FALSE AND
												stDataIn.iDataIn.8 = FALSE AND
													stDataIn.iDataIn.9 = FALSE AND
														stDataIn.iDataIn.10 = FALSE AND
															stDataIn.iDataIn.11 = FALSE AND
																stDataIn.iDataIn.12 = FALSE AND
																	stDataIn.iDataIn.13 = FALSE AND
																		stDataIn.iDataIn.14 = FALSE AND
																			stDataIn.iDataIn.15 = FALSE AND
																				stDataIn.usiState = 159 AND
																					stDataOut.iDataOut = 16#0000 THEN
				//Check if the value is writen in register 31
				stDataOut.usiControl.0 := TRUE;
					stDataOut.usiControl.1 := TRUE;
						stDataOut.usiControl.2 := TRUE;
							stDataOut.usiControl.3 := TRUE;
								stDataOut.usiControl.4 := TRUE;
									stDataOut.usiControl.5 := FALSE;				
										stDataOut.usiControl.6 := FALSE;
											stDataOut.usiControl.7 := TRUE;
												bCheck := TRUE;	
				END_IF	
					
					//Feedback from Input data for register access								
					IF stDataIn.iDataIn.0 = FALSE AND
						stDataIn.iDataIn.1 = FALSE AND
							stDataIn.iDataIn.2 = FALSE AND
								stDataIn.iDataIn.3 = FALSE AND
									stDataIn.iDataIn.4 = FALSE AND
										stDataIn.iDataIn.5 = FALSE AND
											stDataIn.iDataIn.6 = FALSE AND
												stDataIn.iDataIn.7 = FALSE AND
													stDataIn.iDataIn.8 = FALSE AND
														stDataIn.iDataIn.9 = FALSE AND
															stDataIn.iDataIn.10 = FALSE AND
																stDataIn.iDataIn.11 = FALSE AND
																	stDataIn.iDataIn.12 = FALSE AND
																		stDataIn.iDataIn.13 = FALSE AND
																			stDataIn.iDataIn.14 = FALSE AND
																				stDataIn.iDataIn.15 = FALSE AND
																					stDataIn.usiState = 159 THEN 
						eStep := E_Step_Config_Terminal_KL320x.eReadConfiguration_KL320x;
					END_IF	
								
	E_Step_Config_Terminal_KL320x.eReadConfiguration_KL320x:	//Read configuration from register 32
	
		bConfigModeAktiv := TRUE;
			timTimout.IN := TRUE;
				bError := FALSE;

					stDataOut.usiControl.0 := FALSE;
						stDataOut.usiControl.1 := FALSE;
							stDataOut.usiControl.2 := FALSE;
								stDataOut.usiControl.3 := FALSE;
									stDataOut.usiControl.4 := FALSE;
										stDataOut.usiControl.5 := TRUE;				
											stDataOut.usiControl.6 := FALSE;
												stDataOut.usiControl.7 := TRUE;

						//2 wire technic actice or not
						IF stDataIn.iDataIn.10 THEN
								b2Wire := TRUE;
						ELSE	b2Wire := FALSE;						
						END_IF
								
						//Evaluate the sensor type
						IF NOT stDataIn.iDataIn.12 AND NOT stDataIn.iDataIn.13 AND NOT stDataIn.iDataIn.14 AND NOT stDataIn.iDataIn.15 AND stDataIn.usiState = 160 THEN
							sSensorType := 'PT100';
								eStep := E_Step_Config_Terminal_KL320x.eInit_KL320x;
						END_IF
			
						IF NOT stDataIn.iDataIn.12 AND stDataIn.iDataIn.13 AND NOT stDataIn.iDataIn.14 AND NOT stDataIn.iDataIn.15 AND stDataIn.usiState = 160 THEN
							sSensorType := 'PT1000';
								eStep := E_Step_Config_Terminal_KL320x.eInit_KL320x;
						END_IF						
			
						IF NOT stDataIn.iDataIn.12 AND stDataIn.iDataIn.13 AND NOT stDataIn.iDataIn.14 AND NOT stDataIn.iDataIn.15 AND stDataIn.usiState = 160 AND b2Wire THEN
							sSensorType := 'PT100 2 Wire';
								eStep := E_Step_Config_Terminal_KL320x.eInit_KL320x;
						END_IF
								
						IF stDataIn.iDataIn.12 AND stDataIn.iDataIn.13 AND NOT stDataIn.iDataIn.14 AND NOT stDataIn.iDataIn.15 AND stDataIn.usiState = 160 THEN
							sSensorType := 'PT500';
								eStep := E_Step_Config_Terminal_KL320x.eInit_KL320x;
						END_IF
								
						IF NOT stDataIn.iDataIn.12 AND NOT stDataIn.iDataIn.13 AND stDataIn.iDataIn.14 AND NOT stDataIn.iDataIn.15 AND stDataIn.usiState = 160 THEN
							sSensorType := 'PT200';
								eStep := E_Step_Config_Terminal_KL320x.eInit_KL320x;
						END_IF
								
						IF stDataIn.iDataIn.12 AND NOT stDataIn.iDataIn.13 AND NOT stDataIn.iDataIn.14 AND NOT stDataIn.iDataIn.15 AND stDataIn.usiState = 160 THEN
							sSensorType := 'NI100';
								eStep := E_Step_Config_Terminal_KL320x.eInit_KL320x;
						END_IF
								
						IF stDataIn.iDataIn.12 AND NOT stDataIn.iDataIn.13 AND stDataIn.iDataIn.14 AND NOT stDataIn.iDataIn.15 AND stDataIn.usiState = 160 THEN
							sSensorType := 'NI1000';
								eStep := E_Step_Config_Terminal_KL320x.eInit_KL320x;
						END_IF
								
						IF NOT stDataIn.iDataIn.12 AND stDataIn.iDataIn.13 AND stDataIn.iDataIn.14 AND NOT stDataIn.iDataIn.15 AND stDataIn.usiState = 160 THEN
							sSensorType := 'NI120';
								eStep := E_Step_Config_Terminal_KL320x.eInit_KL320x;
						END_IF
								
						IF NOT stDataIn.iDataIn.12 AND stDataIn.iDataIn.13 AND stDataIn.iDataIn.14 AND stDataIn.iDataIn.15 AND stDataIn.usiState = 160 THEN
							sSensorType := 'Resistor from 10Ohm to 5000Ohm';
								eStep := E_Step_Config_Terminal_KL320x.eInit_KL320x;
						END_IF
								
						IF stDataIn.iDataIn.12 AND stDataIn.iDataIn.13 AND stDataIn.iDataIn.14 AND stDataIn.iDataIn.15 AND stDataIn.usiState = 160 THEN
							sSensorType := 'Resistor from 10Ohm to 1200Ohm';
								eStep := E_Step_Config_Terminal_KL320x.eInit_KL320x;
						END_IF
				
END_CASE

	//Timer for Timeout

	timTimout(IN:= , PT:=(T#1S * iTimeout), Q=> , ET=> );
	
	//If we have a timout seth the error bit and go back to the Init step
	IF timTimout.Q THEN
		bError := TRUE;	
			eStep := E_Step_Config_Terminal_KL320x.eInit_KL320x;
	END_IF

END_FUNCTION_BLOCK

// ---- Sensors/FBs Internal/Temperature/FB_TempSensor_M50_P200.TcPOU
{attribute 'hide_all_locals'}
{attribute 'conditionalshow'}
FUNCTION_BLOCK FB_TempSensor_M50_P200
VAR_INPUT
	{attribute 'hide'}
	bEnable							: BOOL;							//Enable or dissable the function
	{attribute 'hide'}
	bUseFilter						: BOOL;							//True = Output Value is filtered, False = Output Value = Raw Input value
	{attribute 'hide'}
	bErrorConfig					: BOOL;							//Error from the config function
	{attribute 'hide'}
	bErrorGeneral					: BOOL;							//Extern general Error
	{attribute 'hide'}
	bWarning						: BOOL;							//Extern general Warning
	{attribute 'hide'}
	bWriteWithDelay					: BOOL;							//Write with Delay the Data to the output (Not al Output Data is writen with Delay)
	{attribute 'hide'}
	usiState						: USINT;						//State from the terminal
	{attribute 'hide'}
	iDelayFilter					: INT := 100;					//Messurement delay in ms
	{attribute 'hide'}
	iMaxValuesFilter				: INT := 10;					//Maximal count of values, max 1000
	{attribute 'hide'}
	iErrorCode						: INT;							//Error Code from external Temperature
	{attribute 'hide'}
	iWarningCode					: INT;							//Warning Code from external Temperature
	{attribute 'hide'}
	rTemperatureOffset				: REAL;							//Temperatur Offset (-10 to +10)
	{attribute 'hide'}
	rRawTempIn						: REAL;							//Temperature raw input value
	{attribute 'hide'}
	tTimDelayOutput					: TIME := T#5S;					//Delay Time to write some Data to the Output
END_VAR
VAR_OUTPUT
	{attribute 'hide'}
	stDataTempOut					: ST_Temperature_Output;		//Temperature output data
	{attribute 'hide'}
	stDataTempOutDelay				: ST_Temperature_Output;		//Temperature output data with delay
END_VAR
VAR
	Filter							: FB_Filter;					//FB Filter for filtering the input value
	timDelayOutputs					: TON;							//Timer to send Data with Delay to the outputs
	FPEnable						: R_TRIG;						//Internal positive Edge
	FNEnable						: F_TRIG;						//Internal negative Edge
END_VAR

//Creator : Kai Ebensperger
//Company : Lynus AG
//Date : 02.06.2021
//Version : 1.0.0.0

//With this function block is possible to realize a temperature senor on the plc
//Work on temperature range from -50°C to 200°C

(*---------------------------------------------------------------Check the limits of the inputs-------------------------------------------------------------------------------*)

iDelayFilter := LIMIT(10,iDelayFilter,10000);
	iMaxValuesFilter := LIMIT(10,iMaxValuesFilter,1000);
		rTemperatureOffset := LIMIT(-10,rTemperatureOffset,10);
			rRawTempIn := LIMIT(-50,rRawTempIn,200);

(*---------------------------------------------------------------Filter the input value-------------------------------------------------------------------------------*)			

Filter(x:= rRawTempIn, tm:= iDelayFilter, k:= iMaxValuesFilter, tbase:= T#1MS, y=> );

IF bUseFilter THEN
	stDataTempOut.rTemperature := Filter.y;	
ELSE
	stDataTempOut.rTemperature := rRawTempIn;
END_IF

(*---------------------------------------------------------------Adjust the sensor value with the offset-------------------------------------------------------------------------------*)

IF rTemperatureOffset <> 0 THEN
	stDataTempOut.rTemperature := stDataTempOut.rTemperature + rTemperatureOffset;
END_IF
	IF rTemperatureOffset = 0 THEN
		stDataTempOut.rTemperature := stDataTempOut.rTemperature;
	END_IF
		
(*---------------------------------------------------------------Error and Warning-------------------------------------------------------------------------------*)

stDataTempOut.byErrorWarning := 0;
	IF bWarning THEN stDataTempOut.byErrorWarning := 1; END_IF  
	IF usiState.0 OR usiState.1 OR usiState.6 OR bErrorConfig OR bErrorGeneral THEN stDataTempOut.byErrorWarning := 2; END_IF	

//Messages and Error Codes
IF stDataTempOut.byErrorWarning = 1 AND iWarningCode = 0 THEN stDataTempOut.eMessage := E_Message_Temperature.eNoConnectionToBackend; 
ELSIF stDataTempOut.byErrorWarning = 2 AND usiState.6 THEN stDataTempOut.eMessage := E_Message_Temperature.eTemperatureGeneralError;
ELSIF stDataTempOut.byErrorWarning = 2 AND usiState.0 THEN stDataTempOut.eMessage := E_Message_Temperature.eTemperatureUnderrangeError;
ELSIF stDataTempOut.byErrorWarning = 2 AND usiState.1 THEN stDataTempOut.eMessage := E_Message_Temperature.eTemperatureOverrangeError;
ELSIF stDataTempOut.byErrorWarning = 2 AND bErrorConfig THEN stDataTempOut.eMessage := E_Message_Temperature.eTemperatureConfigError;	
ELSIF stDataTempOut.byErrorWarning = 2 AND iErrorCode = 0 AND bErrorGeneral THEN stDataTempOut.eMessage := E_Message_Temperature.eTooMuchTemperature;	
ELSE stDataTempOut.eMessage := E_Message_Temperature.eNoMessage; 
END_IF

(*---------------------------------------------------------------Enable-------------------------------------------------------------------------------*)

stDataTempOut.bEnabled := bEnable;
	IF NOT bEnable THEN stDataTempOut.rTemperature := 0; END_IF
	
(*---------------------------------------------------------------Output-------------------------------------------------------------------------------*)

timDelayOutputs(IN:= bWriteWithDelay AND bEnable AND NOT timDelayOutputs.Q, PT:= tTimDelayOutput, Q=> , ET=> );
	FPEnable(CLK:= bEnable, Q=> );
		FNEnable(CLK:= bEnable, Q=> );

stDataTempOut.rTemperature := DINT_TO_REAL(REAL_TO_DINT(stDataTempOut.rTemperature * 100)) / 100;

//Write with Delay or without
IF (bWriteWithDelay AND (timDelayOutputs.Q OR FPEnable.Q OR FNEnable.Q)) OR NOT bWriteWithDelay THEN
	stDataTempOutDelay := stDataTempOut;
END_IF

END_FUNCTION_BLOCK
